// TIA Portal V17 export
// export: Created 2022-07-16T16:56:13.2756588Z, ExportSetting WithDefaults, DisplayName Totally Integrated Automation Portal, DisplayVersion V17, DisplayName TIA Portal Openness, DisplayVersion V17, DisplayName TIA Portal Version Control Interface, DisplayVersion V17, DisplayName TIA Portal Test Suite Advanced, DisplayVersion V17, DisplayName STEP 7 Professional, DisplayVersion V17, DisplayName STEP 7 Safety, DisplayVersion V17, DisplayName WinCC Professional, DisplayVersion V17
TYPE "Client interface_1.dbData.postTestResult.preTestCheckSequence"
// stored: IsFailsafeCompliant false
   STRUCT
      pressures { ExternalWritable := 'False'; S7_SetPoint := 'True'} : "Client interface_1.dbData.postTestResult.preTestCheckSequence.pressures";
   END_STRUCT;
END_TYPE
